Yaskawa INFORM job: TEST-TCP-OFFLINE.JBI

/JOB
//NAME TEST-TCP-OFFLINE
//POS
///NPOS 36,36,36,0,0,0
///TOOL 0
///POSTYPE PULSE
///PULSE
C00000=-3258,-132630,-129331,2447,86477,9228
C00001=-34257,-33510,-74675,-63053,107029,79103
C00002=-69774,-15151,-61825,-51865,89155,72669
C00003=-34257,-33510,-74675,-63053,107029,79103
C00004=-35010,-126399,-87518,-85467,49027,90646
C00005=-46557,-62562,-84163,-57364,51760,71642
C00006=-24386,-85293,-94888,-69954,63152,77974
C00007=-67827,-153552,-117062,-78637,26265,84611
C00008=-81677,-127062,-109504,-49414,21211,70219
C00009=-69876,-155621,-113893,-84716,24272,87496
C00010=-115336,155482,98680,-33462,38477,64065
C00011=-115336,155480,126345,-33462,34267,4503
C00012=-119753,133554,92359,-4505,68534,-1998
C00013=-119235,131828,93963,-4793,66693,-1739
C00014=-119199,119700,69142,-4573,75709,-2076
C00015=-119199,119697,69144,-4573,75711,-2076
C00016=-119251,116954,74052,-4648,71290,-1928
C00017=-119236,117572,62420,-4508,78743,-2201
C00018=-119236,117572,62420,-4508,78743,-2201
C00019=-10120,117572,62420,-4508,78743,-2201
C00020=-10120,117572,62420,-4508,78743,-2201
C00021=-12400,-140475,-135611,-4508,78743,-2201
C00022=-23656,-132888,-133558,-13950,90433,34326
C00023=-29643,-124458,-129653,-12980,91349,32211
C00024=-33108,-115758,-131608,-12491,96374,30552
C00025=-98590,100296,41129,1967,96900,10088
C00026=-100731,130730,83581,2447,86477,9228
C00027=-64686,134954,83581,2447,86477,9228
C00028=-63516,-132630,-129331,2447,86477,9228
C00029=-3258,-132630,-129331,2447,86477,9228
C00030=3,-33511,-74674,-63053,107030,79103
C00031=-65779,-21720,-40488,-89407,90427,72050
C00032=-61888,-62039,-65145,-89619,92976,74681
C00033=-61888,-62039,-65145,-89619,92976,74681
C00034=-85058,56522,31659,-80040,98521,80042
C00035=-52662,-23069,-26207,-57280,52170,72783
BC00000=332203,706510,1050145
BC00001=376793,722392,202725
BC00002=376793,722392,202725
BC00003=381750,742612,222906
BC00004=252867,718865,917690
BC00005=252867,718865,917690
BC00006=252867,718865,917690
BC00007=4169,718865,917690
BC00008=4169,718865,917690
BC00009=4169,718865,917690
BC00010=393877,718866,1061713
BC00011=393877,814209,1061712
BC00012=393877,848513,1061712
BC00013=393877,854433,1050148
BC00014=393877,854433,1050148
BC00015=24253,854433,1050145
BC00016=24253,860833,1050145
BC00017=24253,860833,1050145
BC00018=24253,697829,1050145
BC00019=24253,697829,1050145
BC00020=24253,697829,1050145
BC00021=24253,697829,1050145
BC00022=315293,820005,1050145
BC00023=315293,820005,1050145
BC00024=315293,820005,1050145
BC00025=315293,685500,1050145
BC00026=332203,809604,1050145
BC00027=332203,706510,1050145
BC00028=332203,706510,1050145
BC00029=332203,706510,1050145
BC00030=263565,664642,648758
BC00031=389959,720951,984294
BC00032=389959,720951,984294
BC00033=389884,688585,984294
BC00034=394265,755032,364175
BC00035=27727,677838,524853
EC00000=798157,0
EC00001=-1,0
EC00002=-1,0
EC00003=-1,0
EC00004=-1,0
EC00005=-1,0
EC00006=-1,0
EC00007=-1,0
EC00008=-1,0
EC00009=-1,0
EC00010=0,0
EC00011=0,0
EC00012=0,0
EC00013=0,0
EC00014=0,0
EC00015=0,0
EC00016=0,0
EC00017=0,0
EC00018=0,0
EC00019=0,0
EC00020=798157,0
EC00021=798157,0
EC00022=798157,0
EC00023=798157,0
EC00024=798157,0
EC00025=798157,0
EC00026=798157,0
EC00027=798157,0
EC00028=798157,0
EC00029=798157,0
EC00030=1,-556476
EC00031=1,-556476
EC00032=1,-556476
EC00033=1,-556476
EC00034=4214,-6061
EC00035=4598,-556476
//INST
///DATE 2024/01/25 20:05
///ATTR SC,RW
///GROUP1 RB1,BS1
///GROUP2 ST1
NOP
MOVJ C00000 BC00000 VJ=100.00  +MOVJ EC00000 VJ=100.00
MOVJ C00001 BC00001 VJ=100.00  +MOVJ EC00001 VJ=100.00
'P1
SMOVL C00002 BC00002 V=8.3  +MOVJ EC00002
MOVJ C00003 BC00003 VJ=100.00  +MOVJ EC00003 VJ=100.00
MOVJ C00004 BC00004 VJ=100.00  +MOVJ EC00004 VJ=100.00
'P2
SMOVL C00005 BC00005 V=8.3  +MOVJ EC00005
MOVJ C00006 BC00006 VJ=100.00  +MOVJ EC00006 VJ=100.00
MOVJ C00007 BC00007 VJ=100.00  +MOVJ EC00007 VJ=100.00
'P3
SMOVL C00008 BC00008 V=8.3  +MOVJ EC00008
MOVJ C00009 BC00009 VJ=100.00  +MOVJ EC00009 VJ=100.00
MOVJ C00010 BC00010 VJ=100.00  +MOVJ EC00010 VJ=100.00
MOVJ C00011 BC00011 VJ=100.00  +MOVJ EC00011 VJ=100.00
MOVJ C00012 BC00012 VJ=100.00  +MOVJ EC00012 VJ=100.00
'P4
SMOVL C00013 BC00013 V=8.3  +MOVJ EC00013
MOVJ C00014 BC00014 VJ=100.00  +MOVJ EC00014 VJ=100.00
MOVJ C00015 BC00015 VJ=100.00  +MOVJ EC00015 VJ=100.00
'P5
SMOVL C00016 BC00016 V=8.3  +MOVJ EC00016
MOVJ C00017 BC00017 VJ=100.00  +MOVJ EC00017 VJ=100.00
MOVJ C00018 BC00018 VJ=100.00  +MOVJ EC00018 VJ=100.00
MOVJ C00019 BC00019 VJ=100.00  +MOVJ EC00019 VJ=100.00
MOVJ C00020 BC00020 VJ=100.00  +MOVJ EC00020 VJ=100.00
MOVJ C00021 BC00021 VJ=100.00  +MOVJ EC00021 VJ=100.00
MOVJ C00022 BC00022 VJ=100.00  +MOVJ EC00022 VJ=100.00
'P6
SMOVL C00023 BC00023 V=8.3  +MOVJ EC00023
MOVJ C00024 BC00024 VJ=100.00  +MOVJ EC00024 VJ=100.00
MOVJ C00025 BC00025 VJ=100.00  +MOVJ EC00025 VJ=100.00
'P7
SMOVL C00026 BC00026 V=8.3  +MOVJ EC00026
MOVJ C00027 BC00027 VJ=100.00  +MOVJ EC00027 VJ=100.00
MOVJ C00028 BC00028 VJ=100.00  +MOVJ EC00028 VJ=100.00
MOVJ C00029 BC00029 VJ=100.00  +MOVJ EC00029 VJ=100.00
MOVJ C00030 BC00030 VJ=100.00  +MOVJ EC00030 VJ=100.00
MOVJ C00031 BC00031 VJ=100.00  +MOVJ EC00031 VJ=100.00
'P8
SMOVL C00032 BC00032 V=8.3  +MOVJ EC00032
MOVJ C00033 BC00033 VJ=100.00  +MOVJ EC00033 VJ=100.00
'P9
SMOVL C00034 BC00034 V=8.3  +MOVJ EC00034
'P10
SMOVL C00035 BC00035 V=8.3  +MOVJ EC00035
END
